# EPICS autosave request: tpx3App/Db/ADTimePix_settings.req
file "ADBase_settings.req", P=$(P),  R=$(R)
